// LS Electric XG5000 project: INV_485_MODBUS통신테스트
// PLC NewPLC

PROGRAM Test_Program_1 (task: 스캔 프로그램)

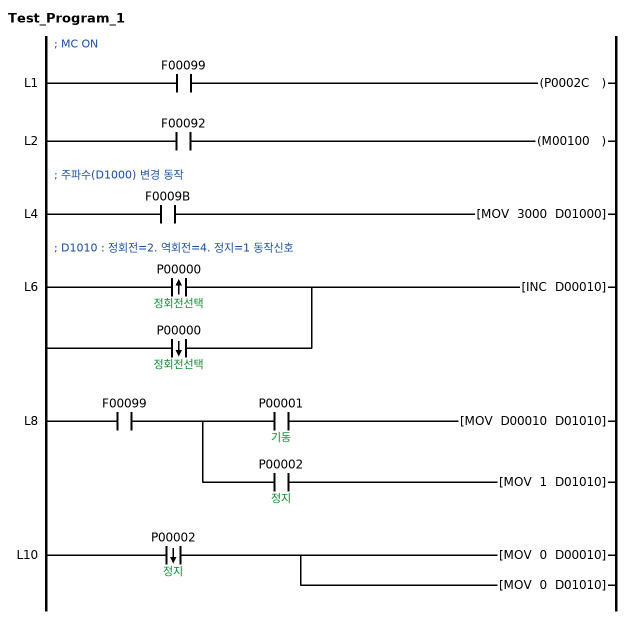
// MC ON
; L1
LOAD      F00099
OUT       P0002C
; L2
LOAD      F00092
OUT       M00100
// 주파수(D1000) 변경 동작
; L4
LOAD      F0009B
MOV       3000 D01000
// D1010 : 정회전=2. 역회전=4. 정지=1 동작신호
; L6
LOADP     P00000	// 정회전선택
ORN       P00000	// 정회전선택
INC       D00010
; L8
LOAD      F00099
MPUSH
AND       P00001	// 기동
MOV       D00010 D01010
MPOP
AND       P00002	// 정지
MOV       1 D01010
; L10
LOADN     P00002	// 정지
MOV       0 D00010
MOV       0 D01010